// TIA Portal V15.1 export
// export: Created 2024-06-21T08:41:02.3979728Z, ExportSetting WithDefaults, DisplayName Totally Integrated Automation Portal, DisplayVersion V15.1 Update 5, DisplayName TIA Portal Openness, DisplayVersion V15.1 Update 5, DisplayName SINAMICS Startdrive Advanced, DisplayVersion V15.1, DisplayName G130, G150, S120, S150, SINAMICS MV, S210, DisplayVersion V15.1, DisplayName G110M, G120, G120C, G120D, G120P, DisplayVersion V15.1, DisplayName STEP 7 Professional, DisplayVersion V15.1 Update 5, DisplayName STEP 7 Safety, DisplayVersion V15.1, DisplayName WinCC Professional, DisplayVersion V15.1 Update 5, DisplayName SIMATIC Visualization Architect, DisplayVersion V15.1
FUNCTION_BLOCK "LProcObjectMode"   // FB1715, FBD
TITLE = LProcObjectMode
{ S7_Optimized_Access := 'FALSE' }
AUTHOR : VCC
FAMILY : ProcEq
NAME : LProcMod
VERSION : 0.1
// ===============================================================================
// This module handles the modes of the process equipments.
// ===============================================================================
// stored: AutoNumber false, IsIECCheckEnabled false, SetENOAutomatically False, UDAEnableTagReadback false
   VAR_INPUT
      I_StartPB { ExternalAccessible := 'False'; ExternalVisible := 'False'; ExternalWritable := 'False'} : Bool;   // Summary Start PB's
      I_EnableAlarm { ExternalAccessible := 'False'; ExternalVisible := 'False'; ExternalWritable := 'False'} : Bool;   // Enable Alarm for the Acof detections
      I_AlarmResetPB { ExternalAccessible := 'False'; ExternalVisible := 'False'; ExternalWritable := 'False'} : Bool;   // Alarm reset pushbutton is activated
      I_GeneralAutoSel { ExternalAccessible := 'False'; ExternalVisible := 'False'; ExternalWritable := 'False'} : Bool;   // General Auto Selection Request
      I_AlarmA { ExternalAccessible := 'False'; ExternalVisible := 'False'; ExternalWritable := 'False'} : Bool;   // Summation Alarm A of roller.
      I_AlarmB { ExternalAccessible := 'False'; ExternalVisible := 'False'; ExternalWritable := 'False'} : Bool;   // Summation Alarm B of roller.
      I_UpperLevelAlarmA { ExternalAccessible := 'False'; ExternalVisible := 'False'; ExternalWritable := 'False'} : Bool;   // Alarm A active from the top level
      I_UpperLevelAlarmB { ExternalAccessible := 'False'; ExternalVisible := 'False'; ExternalWritable := 'False'} : Bool;   // Alarm B active from the top level
      H_HMIModeCmd : Word;   // Mode commands from HMI
   END_VAR
   VAR_OUTPUT
      O_AutoMode { ExternalAccessible := 'False'; ExternalVisible := 'False'; ExternalWritable := 'False'} : Bool;   // Auto mode
      O_ManualMode { ExternalAccessible := 'False'; ExternalVisible := 'False'; ExternalWritable := 'False'} : Bool;   // Manual mode
      O_AutoModeSel { ExternalAccessible := 'False'; ExternalVisible := 'False'; ExternalWritable := 'False'} : Bool;   // Auto Mode Selected
      O_ManualModeSel { ExternalAccessible := 'False'; ExternalVisible := 'False'; ExternalWritable := 'False'} : Bool;   // Manual Mode Selected
      O_ForcedMan { ExternalAccessible := 'False'; ExternalVisible := 'False'; ExternalWritable := 'False'} : Bool;   // Manual Forced Active
      O_FncSelInHMI { ExternalAccessible := 'False'; ExternalVisible := 'False'; ExternalWritable := 'False'} : Bool;   // Manual Selection from HMI
      O_OverTimeAutoSelCond { ExternalAccessible := 'False'; ExternalVisible := 'False'; ExternalWritable := 'False'} : Bool;   // Overtime Auto selected condition
      O_OverTimeAutoSel { ExternalAccessible := 'False'; ExternalVisible := 'False'; ExternalWritable := 'False'} : Bool;   // Alarm Overtime Auto selected
      O_HMISetCmd { ExternalAccessible := 'False'; ExternalVisible := 'False'; ExternalWritable := 'False'} : Bool;   // Set Command on HMI
      O_HMIResetCmd { ExternalAccessible := 'False'; ExternalVisible := 'False'; ExternalWritable := 'False'} : Bool;   // Reset Command on HMI
   END_VAR
   VAR DB_SPECIFIC
      AutoMode { ExternalAccessible := 'False'; ExternalVisible := 'False'; ExternalWritable := 'False'} : Bool;   // Auto mode
      ManualMode { ExternalAccessible := 'False'; ExternalVisible := 'False'; ExternalWritable := 'False'} : Bool;   // Manual mode
      AutoModeSel { ExternalAccessible := 'False'; ExternalVisible := 'False'; ExternalWritable := 'False'} : Bool;   // Auto Mode Selected
      ManualModeSel { ExternalAccessible := 'False'; ExternalVisible := 'False'; ExternalWritable := 'False'} : Bool;   // Manual Mode Selected
      ForcedMan { ExternalAccessible := 'False'; ExternalVisible := 'False'; ExternalWritable := 'False'} : Bool;   // Forced manual active
      H_AutoModeSel { ExternalAccessible := 'False'; ExternalVisible := 'False'; ExternalWritable := 'False'} : Bool;   // Auto Mode Selection from HMI
      H_ManualModeSel { ExternalAccessible := 'False'; ExternalVisible := 'False'; ExternalWritable := 'False'} : Bool;   // Manual Mode Selection from HMI
      H_FncSelInHMI { ExternalAccessible := 'False'; ExternalVisible := 'False'; ExternalWritable := 'False'} : Bool;   // Manual selection from HMI
      H_ForcedMan { ExternalAccessible := 'False'; ExternalVisible := 'False'; ExternalWritable := 'False'} : Bool;   // Forced manual from HMI
      OvTimeAutoSel { ExternalAccessible := 'False'; ExternalVisible := 'False'; ExternalWritable := 'False'} : Bool;   // Alarm Overtime Auto selected and Component activated
      EdgeForceMan { ExternalAccessible := 'False'; ExternalVisible := 'False'; ExternalWritable := 'False'} : Bool;   // Edge Forced Manual from HMI
      ResetForcedMan { ExternalAccessible := 'False'; ExternalVisible := 'False'; ExternalWritable := 'False'} : Bool;   // Reset Forced Manual
      ForcedManTimer { ExternalAccessible := 'False'; ExternalVisible := 'False'; ExternalWritable := 'False'} : Bool;   // Forced manual timer
   END_VAR
   VAR
      TimerOvtAutoSel { ExternalAccessible := 'False'; ExternalVisible := 'False'; ExternalWritable := 'False'; S7_SetPoint := 'True'} : "LTimer";   // Timer Overtime Auto Selected
      TimerForcedMan { ExternalAccessible := 'False'; ExternalVisible := 'False'; ExternalWritable := 'False'; S7_SetPoint := 'True'} : "LTimer";   // Timer Manual Forced
      OvtAutoSel { ExternalAccessible := 'False'; ExternalVisible := 'False'; ExternalWritable := 'False'; S7_SetPoint := 'True'} : "LProc1AlarmMultiIn";   // Alarm Overtime Auto Selected
   END_VAR
   VAR_TEMP   // added for the SCL form of the ladder/FBD networks
      _w1 : Bool;
   END_VAR
BEGIN

REGION Network 1: **** 1 - Inputs **** Extract the modeselection from HMI
   // Extract the modeselection from HMI
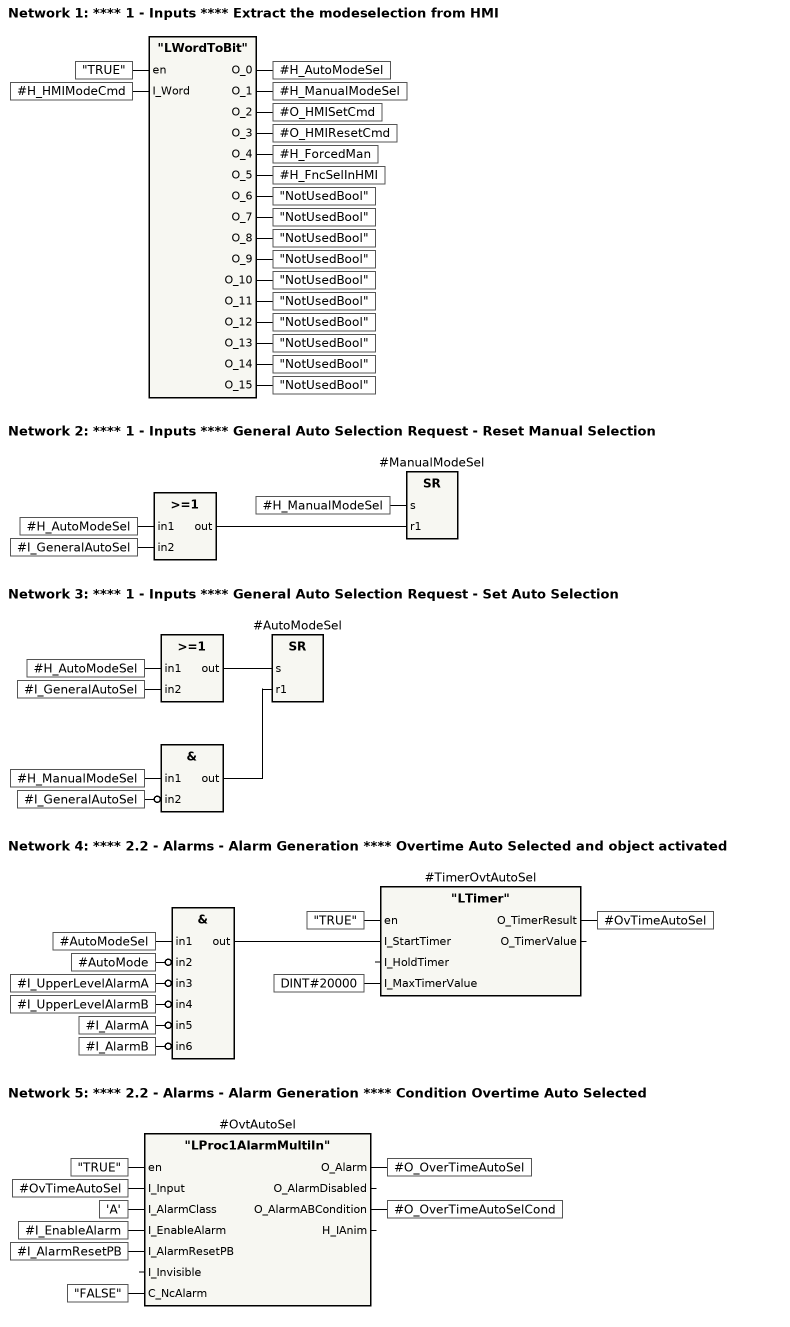
   IF "TRUE" THEN
       "LWordToBit"(I_Word := #H_HMIModeCmd,
                    O_0 => #H_AutoModeSel,
                    O_1 => #H_ManualModeSel,
                    O_2 => #O_HMISetCmd,
                    O_3 => #O_HMIResetCmd,
                    O_4 => #H_ForcedMan,
                    O_5 => #H_FncSelInHMI,
                    O_6 => "NotUsedBool",
                    O_7 => "NotUsedBool",
                    O_8 => "NotUsedBool",
                    O_9 => "NotUsedBool",
                    O_10 => "NotUsedBool",
                    O_11 => "NotUsedBool",
                    O_12 => "NotUsedBool",
                    O_13 => "NotUsedBool",
                    O_14 => "NotUsedBool",
                    O_15 => "NotUsedBool");
   END_IF;
END_REGION

REGION Network 2: **** 1 - Inputs **** General Auto Selection Request - Reset Manual Selection
   // General Auto Selection Request - Reset Manual Selection
   IF #H_ManualModeSel THEN
       #ManualModeSel := TRUE;   // SR flip-flop
   END_IF;
   IF #H_AutoModeSel OR #I_GeneralAutoSel THEN #ManualModeSel := FALSE; END_IF;
END_REGION

REGION Network 3: **** 1 - Inputs **** General Auto Selection Request - Set Auto Selection
   // General Auto Selection Request - Set Auto Selection
   IF #H_AutoModeSel OR #I_GeneralAutoSel THEN
       #AutoModeSel := TRUE;   // SR flip-flop
   END_IF;
   IF #H_ManualModeSel AND NOT #I_GeneralAutoSel THEN #AutoModeSel := FALSE; END_IF;
END_REGION

REGION Network 4: **** 2.2 - Alarms - Alarm Generation **** Overtime Auto Selected and object activated
   // Overtime Auto Selected and object activated
   IF "TRUE" THEN
       #TimerOvtAutoSel(I_StartTimer := #AutoModeSel AND NOT #AutoMode AND NOT #I_UpperLevelAlarmA AND NOT #I_UpperLevelAlarmB AND NOT #I_AlarmA AND NOT #I_AlarmB,   // "LTimer"
                        I_MaxTimerValue := DINT#20000,
                        O_TimerResult => #OvTimeAutoSel);
   END_IF;
END_REGION

REGION Network 5: **** 2.2 - Alarms - Alarm Generation **** Condition Overtime Auto Selected
   // Condition Overtime Auto Selected
   IF "TRUE" THEN
       #OvtAutoSel(I_Input := #OvTimeAutoSel,   // "LProc1AlarmMultiIn"
                   I_AlarmClass := 'A',
                   I_EnableAlarm := #I_EnableAlarm,
                   I_AlarmResetPB := #I_AlarmResetPB,
                   C_NcAlarm := "FALSE",
                   O_Alarm => #O_OverTimeAutoSel,
                   O_AlarmABCondition => #O_OverTimeAutoSelCond);
   END_IF;
END_REGION

REGION Network 6: **** 4.5 - Machine Status - Modes **** Auto mode
   // Auto mode
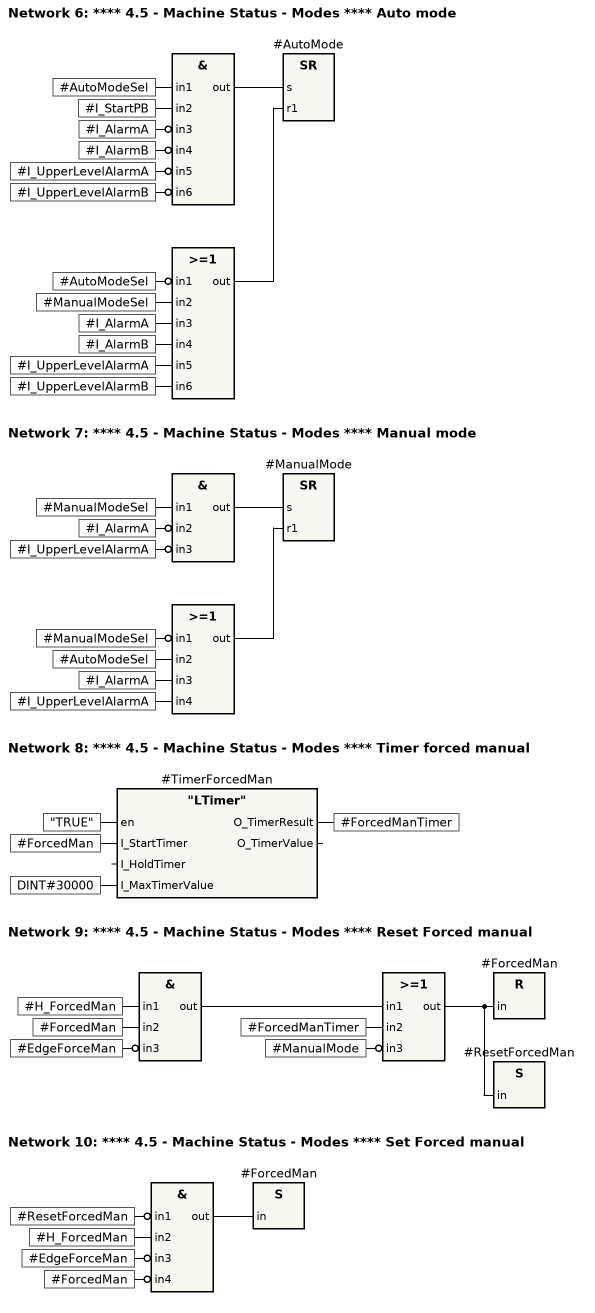
   IF #AutoModeSel AND #I_StartPB AND NOT #I_AlarmA AND NOT #I_AlarmB AND NOT #I_UpperLevelAlarmA AND NOT #I_UpperLevelAlarmB THEN
       #AutoMode := TRUE;   // SR flip-flop
   END_IF;
   IF NOT #AutoModeSel OR #ManualModeSel OR #I_AlarmA OR #I_AlarmB OR #I_UpperLevelAlarmA OR #I_UpperLevelAlarmB THEN
       #AutoMode := FALSE;
   END_IF;
END_REGION

REGION Network 7: **** 4.5 - Machine Status - Modes **** Manual mode
   // Manual mode
   IF #ManualModeSel AND NOT #I_AlarmA AND NOT #I_UpperLevelAlarmA THEN
       #ManualMode := TRUE;   // SR flip-flop
   END_IF;
   IF NOT #ManualModeSel OR #AutoModeSel OR #I_AlarmA OR #I_UpperLevelAlarmA THEN
       #ManualMode := FALSE;
   END_IF;
END_REGION

REGION Network 8: **** 4.5 - Machine Status - Modes **** Timer forced manual
   // Timer forced manual
   IF "TRUE" THEN
       #TimerForcedMan(I_StartTimer := #ForcedMan, I_MaxTimerValue := DINT#30000, O_TimerResult => #ForcedManTimer);   // "LTimer"
   END_IF;
END_REGION

REGION Network 9: **** 4.5 - Machine Status - Modes **** Reset Forced manual
   // Reset Forced manual
   #_w1 := (#H_ForcedMan AND #ForcedMan AND NOT #EdgeForceMan) OR #ForcedManTimer OR NOT #ManualMode;
   IF #_w1 THEN
       #ForcedMan := FALSE;
       #ResetForcedMan := TRUE;
   END_IF;
END_REGION

REGION Network 10: **** 4.5 - Machine Status - Modes **** Set Forced manual
   // Set Forced manual
   IF NOT #ResetForcedMan AND #H_ForcedMan AND NOT #EdgeForceMan AND NOT #ForcedMan THEN
       #ForcedMan := TRUE;
   END_IF;
END_REGION

REGION Network 11: **** 4.5 - Machine Status - Modes **** Set Forced manual
   // Set Forced manual
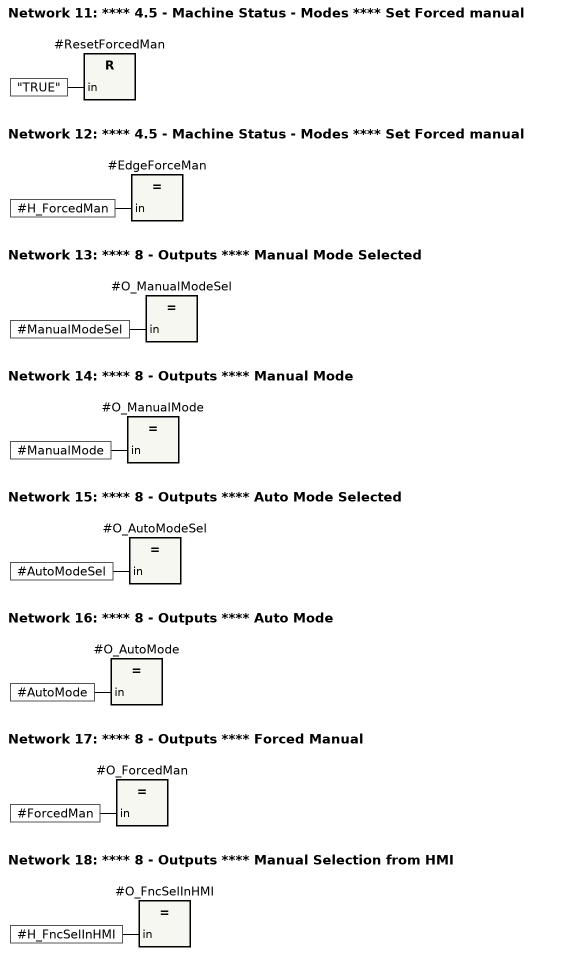
   IF "TRUE" THEN #ResetForcedMan := FALSE; END_IF;
END_REGION

REGION Network 12: **** 4.5 - Machine Status - Modes **** Set Forced manual
   // Set Forced manual
   #EdgeForceMan := #H_ForcedMan;
END_REGION

REGION Network 13: **** 8 - Outputs **** Manual Mode Selected
   // Manual Mode Selected
   #O_ManualModeSel := #ManualModeSel;
END_REGION

REGION Network 14: **** 8 - Outputs **** Manual Mode
   // Manual Mode
   #O_ManualMode := #ManualMode;
END_REGION

REGION Network 15: **** 8 - Outputs **** Auto Mode Selected
   // Auto Mode Selected
   #O_AutoModeSel := #AutoModeSel;
END_REGION

REGION Network 16: **** 8 - Outputs **** Auto Mode
   // Auto Mode
   #O_AutoMode := #AutoMode;
END_REGION

REGION Network 17: **** 8 - Outputs **** Forced Manual
   // Forced Manual
   #O_ForcedMan := #ForcedMan;
END_REGION

REGION Network 18: **** 8 - Outputs **** Manual Selection from HMI
   // Manual Selection from HMI
   #O_FncSelInHMI := #H_FncSelInHMI;
END_REGION
END_FUNCTION_BLOCK
